RoboDK station: BoxSpawner.rdk

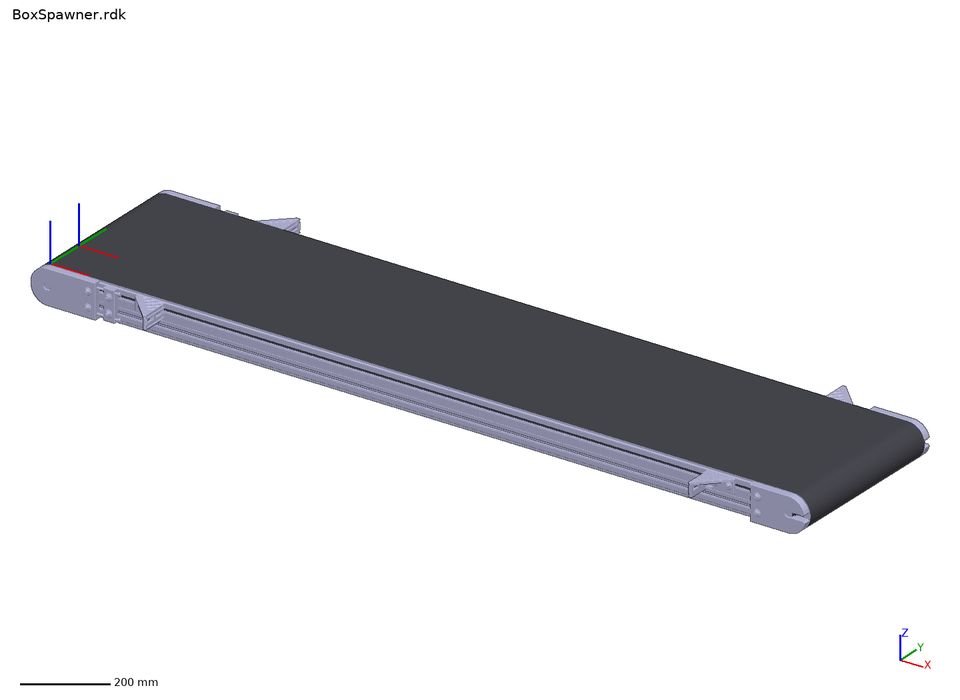
[picture v0: the station drawn from its stored meshes, robots at their saved joint values, targets as dots, program paths as lines]
Station BoxSpawner (saved by RoboDK 5.3.2). Poses are relative to the parent item; angles as X-Y-Z fixed-axis rotations.
Station parameters (name, value as stored): Use Metric, True, BOXSPAWNER_SIZE_X, 200.0, BOXSPAWNER_SIZE_Y, 200.0, BOXSPAWNER_SIZE_Z, 500.0, BOXSPAWNER_UNITS, True, BOXSPAWNER_PARENT, Spawn Location, BOXSPAWNER_CONV_PARENT, Conveyor Frame, BOXSPAWNER_SIZE_X, BOXSPAWNER_SIZE_Y, BOXSPAWNER_SIZE_Z, BOXSPAWNER_UNITS, BOXSPAWNER_PARENT, BOXSPAWNER_CONV_PARENT
  - frame Conveyor Belt Base at (500, 500, 0) mm
    - robot Conveyor Belt: 1 axes
        modified DH rows (alpha deg, a mm, theta deg, d mm): 0, 0, 0, 0 linear
        base shift (0, 0, 0) mm, rotated rx 0 ry 90 rz 0 deg
        joint limits [-500000] to [500000]; home [0]; saved at [0]
      - frame Conveyor Frame at (0, 0, 0) mm
    - frame Spawn Location at (0, 110, 0) mm
  - Python program Spawn Box (listed below)
  - Python program MoveConv (listed below)
  - Python program ResetConv (listed below)
  - program SpawnerLoop (2 instructions, listed below)
  - program Main (3 instructions, listed below)

--- Python program Spawn Box ---
# Type help("robolink") or help("robodk") for more information
# Press F5 to run the script
# Documentation: https://robodk.com/doc/en/RoboDK-API.html
# Reference:     https://robodk.com/doc/en/PythonAPI/index.html
# Note: It is not required to keep a copy of this file, your python script is saved with the station
from robolink import Robolink  # RoboDK API
import SpawnBoxTools as spt

RDK = Robolink()
spt.loadParameters(RDK)
spt.createBox(RDK)

--- Python program MoveConv ---
# Type help("robolink") or help("robodk") for more information
# Press F5 to run the script
# Documentation: https://robodk.com/doc/en/RoboDK-API.html
# Reference:     https://robodk.com/doc/en/PythonAPI/index.html
# Note: It is not required to keep a copy of this file, your python script is saved with the station
from robolink import *  # RoboDK API
from robodk import *  # Robot toolbox

RDK = Robolink()

SPEED = 300  # mm/seconds

conv = RDK.ItemUserPick('Select Conveyor', ITEM_TYPE_ROBOT_AXES)
if not conv.Valid():
    quit()

t = RDK.SimulationTime()
while True:
    s = RDK.SimulationTime() - t
    t = RDK.SimulationTime()

    joints = conv.Joints()
    joints[0] += (SPEED * s)
    conv.setJoints(joints)

    pause(0.001)

--- Python program ResetConv ---
# Type help("robolink") or help("robodk") for more information
# Press F5 to run the script
# Documentation: https://robodk.com/doc/en/RoboDK-API.html
# Reference:     https://robodk.com/doc/en/PythonAPI/index.html
# Note: It is not required to keep a copy of this file, your python script is saved with the station
from robolink import *  # RoboDK API
from robodk import *  # Robot toolbox

RDK = Robolink()

conv = RDK.ItemUserPick('Select Conveyor', ITEM_TYPE_ROBOT_AXES)
if not conv.Valid():
    quit()
conv.setJoints([0])

objects = RDK.ItemList(ITEM_TYPE_OBJECT)
for obj in objects:
    obj.Delete()

--- program SpawnerLoop (robot Conveyor Belt) ---
  Call Spawn Box
  Pause 1.5 s

--- program Main (robot Conveyor Belt) ---
  Call ResetConv
  Run MoveConv
  Call SpawnerLoop
